Staubli VAL3: _resetProgram.pgx

public program _resetProgram()
begin
  if !cycleStatus:bCycle and !cycleStatus:bPause
    if !cycleStatus:bIsHome
      if taskStatus("resetProgram")==-1
          taskCreate "resetProgram",99,gohome:GOHOME()
     //   watch(taskStatus("resetProgram")==1,1)
        wait(taskStatus("resetProgram")==1)
      endIf
    endIf
  endIf
end
